FUNCTION_BLOCK Scale
VAR_INPUT
	EN: BOOL := TRUE;
	x: LREAL;
	x1: LREAL;
	x2: LREAL;
	u1: LREAL;
	u2: LREAL;
END_VAR
VAR_OUTPUT
	ENO: bool;
	u: LREAL;
END_VAR
VAR
END_VAR

IF EN THEN
	IF u1 <= u2 THEN
		u := LimitValue((((x - x1) * (u2 - u1)) / (x2 - x1)) + u1, u1, u2);
	ELSE
		u := LimitValue(u1 - (((x - x1) * (u1 - u2)) / (x2 - x1)), u2, u1);
	END_IF
ELSE
	u := 0;
END_IF
ENO := EN;

END_FUNCTION_BLOCK

(* stored: Version 1.1.0.1, ProductVersion 3.1.4024.3
   POU Scale: Id {79d8db92-1581-43ce-9224-a0c34bb9a397}, SpecialFunc None *)
